{attribute 'qualified_only'}
VAR_GLOBAL CONSTANT
	// One second in microseconds
	OneSecondInUs : UDINT := 1000000;
END_VAR

(* stored: Version 1.1.0.1, ProductVersion 3.1.4022.16
   GVL Constants: Id {7b068a6d-cd30-425d-8e09-2b77bf8b449c} *)
